Fanuc KAREL source: kd00017.KL

-- PROVISIONAL review KL for V1013-1; original PC SHA256 22338fb3581fab95a808a9859f3a233b82dd2acbb813e8f6e76f17d924ba755f
-- Incomplete behavior may be omitted. Consult companion uncertainty JSON. Do not deploy.
PROGRAM KD00017
%NOLOCKGROUP
VAR
  I : INTEGER
  J : INTEGER
  B : BOOLEAN
  R : REAL
  S : STRING[80]
BEGIN
  -- UNRESOLVED_PC offsets 5-12; opcodes 9C,23
  -- UNRESOLVED_PC offsets 17-24; opcodes 22,62
  -- UNRESOLVED_PC offsets 29-36; opcodes 22,28
  -- UNRESOLVED_PC offsets 41-45; opcodes 7F
END KD00017
